RoboDK station: Example-06.c-Pick and place with 2D camera.rdk

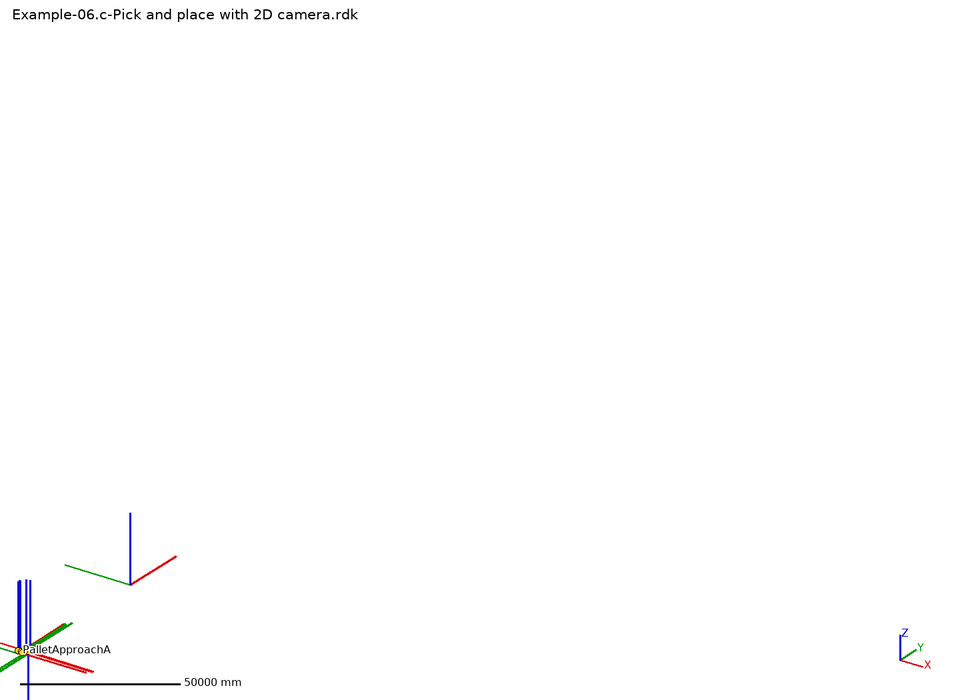
[picture v0: the station drawn from its stored meshes, robots at their saved joint values, targets as dots, program paths as lines]
Station Camera simulation. Poses are relative to the parent item; angles as X-Y-Z fixed-axis rotations.
Station parameters (name, value as stored): SizeBox, 150, 200, 150, SizePallet, 2,3,2, ConvSpeed, 15, SENSOR, 0
  - frame UR10 Base A at (0, -212.57, -10) mm
    - robot UR10 A: 6 axes, payload 10 kg, reach 1300 mm, repeatability 0.1 mm, weight 28.9 kg
        modified DH rows (alpha deg, a mm, theta deg, d mm): 0, 0, 0, 118; 90, 0, 180, 0; 0, 612.7, 0, 0; 0, 571.6, 0, 163.9; -90, 0, 0, 115.7; 90, 0, 180, 92.2
        joint limits [-360, -360, -360, -360, -360, -360] to [360, 360, 360, 360, 360, 360]; home [0, -90, 90, -90, -90, 0]; saved at [165.566, -70.537, 99.931, -119.394, -90, 40.684]
      - tool GripperA, TCP at (0, 0, 30) mm, rotated rx 0 ry 0 rz 90 deg, size 209.9 x 42 x 100 mm, geometry from test.iges
    - frame PalletA at (-344.62, -460.78, -266.49) mm, rotated rx 0 ry 0 rz 90.24 deg
      - object Europallet at (0, 0, 0) mm, size 800 x 144 x 1200 mm, geometry from User Library-Europallet.igs
      - object box100mm at (0, 0, 0) mm, size 100 x 100 x 100 mm, geometry from box.sld
      - object Part 1 at (75, 100, 75) mm, size 150 x 200 x 150 mm, geometry from box.sld
      - object Part 2 at (225, 100, 75) mm, size 150 x 200 x 150 mm, geometry from box.sld
      - object Part 3 at (75, 300, 75) mm, size 150 x 200 x 150 mm, geometry from box.sld
      - object Part 4 at (225, 300, 75) mm, size 150 x 200 x 150 mm, geometry from box.sld
      - object Part 5 at (75, 500, 75) mm, size 150 x 200 x 150 mm, geometry from box.sld
      - object Part 6 at (225, 500, 75) mm, size 150 x 200 x 150 mm, geometry from box.sld
      - object Part 7 at (75, 100, 225) mm, size 150 x 200 x 150 mm, geometry from box.sld
      - object Part 8 at (225, 100, 225) mm, size 150 x 200 x 150 mm, geometry from box.sld
      - object Part 9 at (75, 300, 225) mm, size 150 x 200 x 150 mm, geometry from box.sld
      - object Part 10 at (225, 300, 225) mm, size 150 x 200 x 150 mm, geometry from box.sld
      - object Part 11 at (75, 500, 225) mm, size 150 x 200 x 150 mm, geometry from box.sld
      - object Part 12 at (225, 500, 225) mm, size 150 x 200 x 150 mm, geometry from box.sld
    - target PalletApproachA (joint target) at (-397.36, -413.15, 569.38) mm, rotated rx 180 ry 0 rz 88.83 deg; joints [29.502, -102.797, 97.668, -84.871, -90, -59.329] of UR10 A
    - target ConvApproachA (joint target) at (711.87, -183.71, 533.48) mm, rotated rx -180 ry -0.01 rz 172.23 deg; joints [152.649, -87.247, 87.177, -89.921, -90.005, -19.581] of UR10 A
  - frame UR10 Base B at (1478.64, 1242.75, 0) mm
    - robot UR10 B: 6 axes, payload 10 kg, reach 1300 mm, repeatability 0.1 mm, weight 28.9 kg
        modified DH rows (alpha deg, a mm, theta deg, d mm): 0, 0, 0, 118; 90, 0, 180, 0; 0, 612.7, 0, 0; 0, 571.6, 0, 163.9; -90, 0, 0, 115.7; 90, 0, 180, 92.2
        joint limits [-360, -360, -360, -360, -360, -360] to [360, 360, 360, 360, 360, 360]; home [0, -90, 90, -90, -90, 0]; saved at [-180.64, -99.905, 114.086, -104.182, -90, 0]
      - tool GripperB, TCP at (0, 0, 40) mm, rotated rx 0 ry 0 rz 90 deg, size 209.9 x 42 x 100 mm, geometry from test.iges
      - frame Camera Reference at (78.3, -93.59, 25.69) mm, rotated rx 0 ry 0 rz -90 deg
        - object SICK VSPP-5F2113 at (0, 0, 0) mm, size 53 x 116 x 38 mm, geometry from SICK VSPx.sld
    - target ConvApproachB (joint target) at (-305.88, 88.81, 332.02) mm, rotated rx -180 ry 0 rz 0 deg; joints [-47.16, -132.426, 135.54, -93.114, -90, -47.16] of UR10 B
    - target PalletApproachB (joint target) at (566.28, 157.58, 374.33) mm, rotated rx -180 ry 0 rz 179.36 deg; joints [-180.64, -99.905, 114.086, -104.182, -90, 0] of UR10 B
    - target InspectPartB (joint target) at (-571.45, -82.78, 699.15) mm, rotated rx -180 ry 0 rz 0 deg; joints [-8.247, -99.686, 80.867, -71.181, -90, -8.247] of UR10 B
    - frame PalletB at (1034.81, 598.47, -166.38) mm, rotated rx 0 ry 0 rz 180 deg
      - object Europallet at (0, 0, 0) mm, size 800 x 144 x 1200 mm, geometry from User Library-Europallet.igs
  - frame ConveyorReference at (597.23, -679.82, 119.18) mm
    - robot Conveyor Belt: 1 axes
        modified DH rows (alpha deg, a mm, theta deg, d mm): 0, 0, 0, 0 linear
        base shift (440, 200, 0) mm, rotated rx 0 ry 90 rz 90 deg
        joint limits [-500000] to [500000]; home [0]; saved at [58958]
      - frame MovingRef at (0, 0, 0) mm
    - target ConveyorHome (joint target) at (440, 200, 0) mm, rotated rx 0 ry 0 rz 90 deg; joints [0] of Conveyor Belt
    - target ConveyorMove (joint target) at (440, 500200, 0) mm, rotated rx 0 ry 0 rz 90 deg; joints [500000] of Conveyor Belt
    - target Get Conveyor (Cartesian target) at (200, 1900, 0) mm, rotated rx -180 ry 0 rz 0 deg; joints [-12.012, -77.865, 120.975, -133.11, -90, -12.012] of UR10 B
    - target Put Conveyor (Cartesian target) at (200, 422.12, 0) mm, rotated rx -180 ry 0 rz 180 deg; joints [7.229, -35.446, 107.125, -161.679, -90, 96.985] of UR10 A
  - Python program SetSimulationParams (listed below)
  - Python program PrepareSimulation (listed below)
  - Python program SimulateCamera (listed below)
  - Python program PartsToConveyor (listed below)
  - Python program PartsToPallet (listed below)
  - program MoveConveyor (1 instructions, listed below)
  - program MainSimulation (5 instructions, listed below)

--- Python program SetSimulationParams ---
# Type help("robolink") or help("robodk") for more information
# Press F5 to run the script
# Note: you do not need to keep a copy of this file, your python script is saved with the station
from robolink import *    # API to communicate with RoboDK
from robodk import *      # basic matrix operations


PARAM_SIZE_BOX = 'SizeBox'
PARAM_SIZE_PALLET = 'SizePallet'
PARAM_CONV_SPEED_MM = 'ConvSpeed'



RDK = Robolink()

size_box = RDK.getParam(PARAM_SIZE_BOX)
size_pallet = RDK.getParam(PARAM_SIZE_PALLET)
conv_speed = RDK.getParam(PARAM_CONV_SPEED_MM)

# ------------------------------------------------------------
size_box_input = mbox('Enter the size of the box in mm [L,W,H]', entry=size_box)
if size_box_input:
    RDK.setParam(PARAM_SIZE_BOX, size_box_input)
else:
    raise Exception('Operation cancelled by user')

# ------------------------------------------------------------
size_pallet_input = mbox('Enter the size of the pallet', entry=size_pallet)
if size_pallet_input:
    RDK.setParam(PARAM_SIZE_PALLET, size_pallet_input)
else:
    raise Exception('Operation cancelled by user')

# ------------------------------------------------------------
conv_speed_input = mbox('Enter the speed of the conveyor in mm/s', entry=conv_speed)
if conv_speed_input:
    RDK.setParam(PARAM_CONV_SPEED_MM, conv_speed_input)
    conv_speed = float(conv_speed_input)
    conv = RDK.Item('Conveyor Belt', ITEM_TYPE_ROBOT)
    conv.setSpeed(conv_speed)

else:
    raise Exception('Operation cancelled by user')

--- Python program PrepareSimulation ---
# Type help("robolink") or help("robodk") for more information
# Press F5 to run the script
# Note: you do not need to keep a copy of this file, your python script is saved with the station
from robolink import *    # API to communicate with RoboDK
from robodk import *      # basic matrix operations

# Use RoboDK API as RL
RDK = Robolink()

frame_pallet        = RDK.Item('PalletA', ITEM_TYPE_FRAME)

# get variable parameters
SIZE_BOX = RDK.getParam('SizeBox')
SIZE_PALLET = RDK.getParam('SizePallet')
SIZE_BOX_XYZ = [float(x.replace(' ','')) for x in SIZE_BOX.split(',')]
SIZE_PALLET_XYZ = [float(x.replace(' ','')) for x in SIZE_PALLET.split(',')]
SIZE_BOX_Z = SIZE_BOX_XYZ[2] # the height of the boxes is important to take into account when approaching the positions

def box_calc(size_xyz, pallet_xyz):
    """Calculates a list of points to store parts in a pallet"""
    [size_x, size_y, size_z] = size_xyz
    [pallet_x, pallet_y, pallet_z] = pallet_xyz
    xyz_list = []
    for h in range(int(pallet_z)):
        for j in range(int(pallet_y)):
            for i in range(int(pallet_x)):
                xyz_list = xyz_list + [[(i+0.5)*size_x, (j+0.5)*size_y, (h+0.5)*size_z]]
    return xyz_list

def parts_setup(frame, positions, size_xyz):
    """Place a list of parts in a reference frame. The part/reference object must have been previously copied to the clipboard."""
    [size_x, size_y, size_z] = size_xyz
    nparts = len(positions)
    cstep = 1.0/(nparts - 1)
    for i in range(nparts):
        newpart = frame.Paste()
        newpart.Scale([size_x/100, size_y/100, size_z/100]) #scale with respect to the reference object (100mm cube)
        newpart.setName('Part ' + str(i+1)) #set item name
        newpart.setPose(transl(positions[i])) #set item position with respect to parent
        newpart.setVisible(True, False) #make item visible but hide the reference frame
        newpart.Recolor([1-cstep*i, cstep*i, 0.2, 1]) #set RGBA color

def cleanup(objects, startswith="Part "):
    """Deletes all objects where the name starts with "startswith", from the provided list of objects."""
    for item in objects:
        if item.Name().startswith(startswith):
            item.Delete()

# turn off rendering (much faster when setting up the station)
RDK.Render(False)

# cleanup previous simulation (generated parts and tools)
all_objects = RDK.ItemList(ITEM_TYPE_OBJECT, False)
cleanup(all_objects, 'Part ')
all_tools = RDK.ItemList(ITEM_TYPE_TOOL, False)
cleanup(all_tools, 'TCP ')

# copy the reference part
partref = RDK.Item('box100mm')
partref.Copy()

#RL.Set_Simulation_Speed(500);
#RL.Set_Simulation_Mode(1)

# calculate an array of positions to get/store the parts
parts_positions = box_calc(SIZE_BOX_XYZ, SIZE_PALLET_XYZ)

# setup/initialise the parts on the palled
parts_setup(frame_pallet, parts_positions, SIZE_BOX_XYZ)

RDK.Render(True)

--- Python program SimulateCamera ---
# Type help("robolink") or help("robodk") for more information
# Press F5 to run the script
# Note: you do not need to keep a copy of this file, your python script is saved with the station
from robolink import *    # API to communicate with RoboDK
from robodk import *      # basic matrix operations
RDK = Robolink()

# Close any open 2D camera views
RDK.Cam2D_Close()

camref = RDK.Item('Camera Reference',ITEM_TYPE_FRAME)

# set parameters in mm and degrees:
# FOV: Field of view in degrees (atan(0.5*height/distance) of the sensor divided by
# FOCAL_LENGHT: focal lenght in mm
# FAR_LENGHT: maximum working distance (in mm)
# SIZE: size of the sensor in pixels
# BG_COLOR: background color (rgb color or named color: AARRGGBB)
# LIGHT_AMBIENT: ambient color (rgb color or named color: AARRGGBB)
# LIGHT_SPECULAR: specular color (rgb color or named color: AARRGGBB)
# LIGHT_DIFFUSE: diffuse color (rgb color or named color: AARRGGBB)


# cam_id = RDK.Cam2D_Add(camref, 'FOCAL_LENGHT=6 FOV=32 FAR_LENGHT=1000 SIZE=640x480 BG_COLOR=black')
# cam_id = RDK.Cam2D_Add(camref, 'FOCAL_LENGHT=6 FOV=32 FAR_LENGHT=1000 SIZE=640x480')
# cam_id = RDK.Cam2D_Add(camref, 'FOCAL_LENGHT=6 FOV=32 FAR_LENGHT=1000 SIZE=640x480 BG_COLOR=black LIGHT_AMBIENT=red LIGHT_DIFFUSE=#FF00FF00 LIGHT_SPECULAR=black')
# cam_id = RDK.Cam2D_Add(camref, 'FOCAL_LENGHT=6 FOV=32 FAR_LENGHT=1000 SIZE=640x480 DEPTH')
cam_id = RDK.Cam2D_Add(camref, 'FOCAL_LENGHT=6 FOV=32 FAR_LENGHT=1000 SIZE=640x480 BG_COLOR=black LIGHT_AMBIENT=red LIGHT_DIFFUSE=black LIGHT_SPECULAR=white')


# cam_id = RDK.Cam2D_Add(camref, 'FOCAL_LENGHT=6 FOV=32 FAR_LENGHT=1000 SIZE=640x480 LIGHT_AMBIENT=red')

# cam_id = RDK.Cam2D_Add(camref, 'POPUP')

# RDK.Cam2D_Snapshot(RDK.getParam('PATH_OPENSTATION') + "/sample_image.png", cam_id)

--- Python program PartsToConveyor ---
# Type help("robolink") or help("robodk") for more information
# Press F5 to run the script
# Note: you do not need to keep a copy of this file, your python script is saved with the station
from robolink import *    # API to communicate with RoboDK
from robodk import *      # basic matrix operations
from random import uniform

# Use RoboDK API as RL
RDK = Robolink()

# define default approach distance
APPROACH = 100

# gather robot, tool and reference frames from the station
robot               = RDK.Item('UR10 A', ITEM_TYPE_ROBOT)
tool                = RDK.Item('GripperA', ITEM_TYPE_TOOL)
frame_pallet        = RDK.Item('PalletA', ITEM_TYPE_FRAME)
frame_conv          = RDK.Item('ConveyorReference', ITEM_TYPE_FRAME)
frame_conv_moving   = RDK.Item('MovingRef', ITEM_TYPE_FRAME)

# gather targets
target_pallet_safe = RDK.Item('PalletApproachA', ITEM_TYPE_TARGET)
target_conv_safe = RDK.Item('ConvApproachA', ITEM_TYPE_TARGET)
target_conv = RDK.Item('Put Conveyor', ITEM_TYPE_TARGET)

# get variable parameters
SIZE_BOX = RDK.getParam('SizeBox')
SIZE_PALLET = RDK.getParam('SizePallet')
SIZE_BOX_XYZ = [float(x.replace(' ','')) for x in SIZE_BOX.split(',')]
SIZE_PALLET_XYZ = [float(x.replace(' ','')) for x in SIZE_PALLET.split(',')]
SIZE_BOX_Z = SIZE_BOX_XYZ[2] # the height of the boxes is important to take into account when approaching the positions

def box_calc(size_xyz, pallet_xyz):
    """Calculates a list of points to store parts in a pallet"""
    [size_x, size_y, size_z] = size_xyz
    [pallet_x, pallet_y, pallet_z] = pallet_xyz
    xyz_list = []
    for h in range(int(pallet_z)):
        for j in range(int(pallet_y)):
            for i in range(int(pallet_x)):
                xyz_list = xyz_list + [[(i+0.5)*size_x, (j+0.5)*size_y, (h+0.5)*size_z]]
    return xyz_list

def TCP_On(toolitem):
    """Attaches the closest object to the toolitem Htool pose,
    It will also output appropriate function calls on the generated robot program (call to TCP_On)"""
    toolitem.AttachClosest()
    toolitem.RDK().RunMessage('Set air valve on')
    toolitem.RDK().RunProgram('TCP_On()');

def TCP_Off(toolitem, itemleave=0):
    """Detaches the closest object attached to the toolitem Htool pose,
    It will also output appropriate function calls on the generated robot program (call to TCP_Off)"""
    toolitem.DetachAll(itemleave)
    toolitem.RDK().RunMessage('Set air valve off')
    toolitem.RDK().RunProgram('TCP_Off()');

#RL.Set_Simulation_Speed(500);
#RL.Set_Simulation_Mode(1)

# calculate an array of positions to get/store the parts
parts_positions = box_calc(SIZE_BOX_XYZ, SIZE_PALLET_XYZ)

# Calculate a new TCP that takes into account the size of the part (targets are set to the center of the box)
tool_xyzrpw = tool.PoseTool()*transl(0,0,SIZE_BOX_Z/2)
tool_tcp = robot.AddTool(tool_xyzrpw, 'TCP A')

# ---------------------------------------------------------------------------------
# -------------------------- PROGRAM START ----------------------------------------

robot.setPoseTool(tool_tcp)
nparts = len(parts_positions)
i = nparts-1
while i >= 0:
    # ----------- take a part from the pallet ------
    # get the xyz position of part i
    robot.setPoseFrame(frame_pallet)
    part_position_i = parts_positions[i]
    target_i = transl(part_position_i)*rotx(pi)
    target_i_app = target_i * transl(0,0,-(APPROACH+SIZE_BOX_Z))
    # approach to the pallet
    robot.MoveJ(target_pallet_safe)
    # get the box i
    robot.MoveJ(target_i_app)
    robot.MoveL(target_i)
    TCP_On(tool) # attach the closest part
    robot.MoveL(target_i_app)
    robot.MoveJ(target_pallet_safe)

    # ----------- place the box i on the convegor ------
    # approach to the conveyor
    robot.setPoseFrame(frame_conv)
    target_conv_pose = target_conv.Pose()*transl(0,0,-SIZE_BOX_Z/2)
    target_conv_app = target_conv_pose*transl(0,0,-APPROACH)
    robot.MoveJ(target_conv_safe)
    robot.MoveJ(target_conv_app)

    # Place the part at a random position with respect to the target on the conveyor
    TX = uniform(-150, 150)
    RZ = uniform(-90*pi/180, +90*pi/180)

    robot.MoveL(target_conv_pose*transl(TX,0,0)*rotz(RZ))
    TCP_Off(tool, frame_conv_moving) # detach an place the object in the moving reference frame of the conveyor
    robot.MoveL(target_conv_app)
    robot.MoveJ(target_conv_safe)

    i = i - 1

--- Python program PartsToPallet ---
# Type help("robolink") or help("robodk") for more information
# Press F5 to run the script
# Note: you do not need to keep a copy of this file, your python script is saved with the station
from robolink import *    # API to communicate with RoboDK
from robodk import *      # basic matrix operations

# Use RoboDK API as RL
RDK = Robolink()

# define default approach distance
APPROACH = 100
SENSOR_VARIABLE = 'SENSOR' # station variable
PART_KEYWORD = 'Part' # parts to look for (camera simulation)

# gather robot, tool and reference frames from the station
robot               = RDK.Item('UR10 B', ITEM_TYPE_ROBOT)
tool                = RDK.Item('GripperB', ITEM_TYPE_TOOL)
frame_pallet        = RDK.Item('PalletB', ITEM_TYPE_FRAME)
frame_conv          = RDK.Item('ConveyorReference', ITEM_TYPE_FRAME)
frame_conv_moving   = RDK.Item('MovingRef', ITEM_TYPE_FRAME)

# gather targets
target_pallet_safe = RDK.Item('PalletApproachB', ITEM_TYPE_TARGET)
target_conv_safe = RDK.Item('ConvApproachB', ITEM_TYPE_TARGET)
target_conv = RDK.Item('Get Conveyor', ITEM_TYPE_TARGET)
target_inspect = RDK.Item('InspectPartB', ITEM_TYPE_TARGET)

# get variable parameters
SIZE_BOX = RDK.getParam('SizeBox')
SIZE_PALLET = RDK.getParam('SizePallet')
SIZE_BOX_XYZ = [float(x.replace(' ','')) for x in SIZE_BOX.split(',')]
SIZE_PALLET_XYZ = [float(x.replace(' ','')) for x in SIZE_PALLET.split(',')]
SIZE_BOX_Z = SIZE_BOX_XYZ[2] # the height of the boxes is important to take into account when approaching the positions

camera_ref_conv = target_conv.PoseAbs()

#----------------- camera simulation
# Get all object names to
all_objects = RDK.ItemList(ITEM_TYPE_OBJECT, True)

# Get object items in a list (faster) and filter by keyword
check_objects = []
for i in range(len(all_objects)):
    if all_objects[i].count(PART_KEYWORD) > 0:
        check_objects.append(RDK.Item(all_objects[i]))

# Make sure that there is at least one part that we are expecting
if len(check_objects) == 0:
    raise Exception('No parts to check for. Name at least one part with the name: %s.' % PICKABLE_OBJECTS_KEYWORD)

# simulates the behavior of the camera (returns TX, TY and RZ)
def WaitPartCamera():
    """Simulate camera detection"""
    if RDK.RunMode() == RUNMODE_SIMULATE:
        # Simulate the camera by waiting for an object to be detected
        while True:
            for part in check_objects:
                # calculate the position of the part with respect to the target
                part_pose = invH(camera_ref_conv) * part.PoseAbs()
                tx,ty,tz,rx,ry,rz = pose_2_xyzrpw(part_pose)
                rz = rz * pi/180.0 # Convert degrees to radians
                if abs(tx) < 400 and ty < 50 and abs(tz) < 400:
                    print('Part detected: TX,TY,TZ=%.1f,%.1f,%.1f' % (tx,ty,rz))
                    return tx, ty, rz
            pause(0.005)
    else:
        RDK.RunProgram('WaitPartCamera')
    return 0,0,0

#-----------------------------

def box_calc(size_xyz, pallet_xyz):
    """Calculates a list of points to store parts in a pallet"""
    [size_x, size_y, size_z] = size_xyz
    [pallet_x, pallet_y, pallet_z] = pallet_xyz
    xyz_list = []
    for h in range(int(pallet_z)):
        for j in range(int(pallet_y)):
            for i in range(int(pallet_x)):
                xyz_list = xyz_list + [[(i+0.5)*size_x, (j+0.5)*size_y, (h+0.5)*size_z]]
    return xyz_list

def TCP_On(toolitem):
    """Attaches the closest object to the toolitem Htool pose,
    It will also output appropriate function calls on the generated robot program (call to TCP_On)"""
    toolitem.AttachClosest()
    toolitem.RDK().RunMessage('Set air valve on')
    toolitem.RDK().RunProgram('TCP_On()');

def TCP_Off(toolitem, itemleave=0):
    """Detaches the closest object attached to the toolitem Htool pose,
    It will also output appropriate function calls on the generated robot program (call to TCP_Off)"""
    #toolitem.DetachClosest(itemleave)
    toolitem.DetachAll(itemleave)
    toolitem.RDK().RunMessage('Set air valve off')
    toolitem.RDK().RunProgram('TCP_Off()');

# calculate an array of positions to get/store the parts
parts_positions = box_calc(SIZE_BOX_XYZ, SIZE_PALLET_XYZ)

# Calculate a new TCP that takes into account the size of the part (targets are set to the center of the box)
tool_xyzrpw = tool.PoseTool()*transl(0,0,SIZE_BOX_Z/2)
tool_tcp = robot.AddTool(tool_xyzrpw, 'TCP B')

# ---------------------------------------------------------------------------------
# -------------------------- PROGRAM START ----------------------------------------
robot.setPoseTool(tool_tcp)
nparts = len(parts_positions)
i = 0
while i < nparts:
    # ----------- take a part from the convegor ------
    # approach to the conveyor
    robot.setPoseFrame(frame_conv)
    robot.MoveJ(target_inspect)

    #------------------------- camera simulation
    CAM_TX, CAM_TY, CAM_RZ = WaitPartCamera()
    # Adjust position along movement according to conveyor speed
    CAM_TY = CAM_TY - 50
    # Lazy move: the part is symmetrical so there is no need to turn more than +/-90 deg around the Z axis. If so, add as many half turns as required
    if CAM_RZ > pi/2:
        CAM_RZ = CAM_RZ - pi
    elif CAM_RZ < -pi/2:
        CAM_RZ = CAM_RZ + pi
    target_conv_pose = target_conv.Pose()*transl(CAM_TX,CAM_TY,-SIZE_BOX_Z/2)*rotz(CAM_RZ)
    target_conv_app = target_conv_pose*transl(0,0,-APPROACH)
    #-------------------------------------------------

    robot.MoveL(target_conv_pose)
    TCP_On(tool) # detach an place the object in the moving reference frame of the conveyor
    robot.MoveL(target_conv_app)

    if len(tool.Childs()) == 0:
        # Detect invalid pick
        continue

    robot.MoveJ(target_conv_safe)

    # ----------- place the part on the pallet ------
    # get the xyz position of part i
    robot.setPoseFrame(frame_pallet)
    part_position_i = parts_positions[i]
    target_i = transl(part_position_i)*rotx(pi)
    target_i_app = target_i * transl(0,0,-(APPROACH+SIZE_BOX_Z))
    # approach to the pallet
    robot.MoveJ(target_pallet_safe)
    # get the box i
    robot.MoveJ(target_i_app)
    robot.MoveL(target_i)
    TCP_Off(tool, frame_pallet) # attach the closest part
    robot.MoveL(target_i_app)
    robot.MoveJ(target_pallet_safe)

    i = i + 1

--- program MoveConveyor (robot Conveyor Belt) ---
  MoveJ (ConveyorMove)

--- program MainSimulation (robot UR10 A) ---
  Call PrepareSimulation
  Call SimulateCamera
  Run MoveConveyor
  Run PartsToConveyor
  Call PartsToPallet
